/// calibration that is determined by calibration sequences of the unit (static offsets, shifts)
TYPE MachineDataCalibration :
STRUCT
END_STRUCT
END_TYPE

(* stored: Version 1.1.0.1
   DUT MachineDataCalibration: Id {3cf0e6ef-15c9-4e6d-bdef-f97e7939a724} *)
